(* Logix 5000 project; controller Ex_2_03 Emulate 5570 rev 33.11; software revision 33.00 *)
// Turn off light in lamp with push button

TASK MainTask (continuous, watchdog 500 ms) : MainProgram

MODULES
   Local : Emulate 5570 (ICP 4, rev 33.11)
END_MODULES

VAR_GLOBAL   (* controller tags *)
   P2 : BOOL;   // Lamp_P2
   S2 : BOOL;   // Push Button S2
END_VAR

PROGRAM MainProgram   (* main routine MainRoutine *)

ROUTINE MainRoutine   (* ladder *)
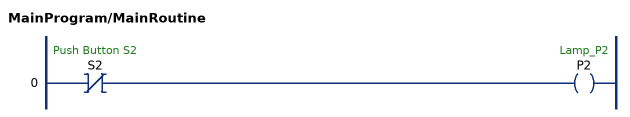
   0: XIO(S2)OTE(P2);
END_ROUTINE
END_PROGRAM
